FUNCTION NotValue : I_BoolValue
VAR_INPUT
	boolean : REFERENCE TO BOOL;
END_VAR
VAR
	p : POINTER TO FB_BoolBindingReadOnly;
END_VAR

p := __NEW(FB_BoolBindingReadOnly);

p^.Bind(boolean);
p^.Negate := TRUE;

NotValue := p^;

END_FUNCTION

(* stored: Version 1.1.0.1
   POU NotValue: Id {809af615-d612-4af0-a510-c79c246103b6}, SpecialFunc None *)
